// Mitsubishi GX Works2 project: PID_slave_FX3U_26_04_2021   PLC: FX3U/FX3UC

// global labels: Global1
VAR_GLOBAL
  anaDig1 AT D8260 : INT;  (* Analog input from AD converter Level transmitter *)
  anaDig2 AT D8261 : INT;  (* Analog input from AD converter Flow transmitter *)
  digAna AT D8262 : INT;  (* Analog output from DA converter Level Vaulve *)
  Pump AT Y000 : BOOL;  (* Kontaktor til drift av pumpe *)
  AlarmLamp AT Y001 : BOOL;  (* Alarm lampe til systemet *)
  MagnetValve_1 AT Y004 : BOOL;  (* Magnetventil 1 *)
  MagnetValve_2 AT Y005 : BOOL;  (* Magnetventil 2 *)
  MagnetValve_3 AT Y006 : BOOL;  (* Magnetventil 3 *)
  Input_OnOff AT M100 : BOOL;  (* On off for the system *)
  Input_ManualMode AT M500 : BOOL;  (* Valg av Manuell "1" eller Auto "0" *)
  Input_OperationModus AT M501 : BOOL;  (* Valg av direkte "1" eller Revers "0" Regulering *)
  Input_IntegratorModus AT M502 : BOOL;  (* Valg av Integrator virkning på regulator *)
  Input_DerivatorModus AT M503 : BOOL;  (* Valg av Derivator virkning på regulator *)
  Input_Pump AT M504 : BOOL;  (* Start signal til pumpe fra Master *)
  Input_AlarmLamp AT M505 : BOOL;  (* Start signal til Alarm lampe fra Master *)
  Input_MagnetValve_1 AT M506 : BOOL;  (* Start signal til Magnetventil 1 fra Master *)
  Input_MagnetValve_2 AT M507 : BOOL;  (* Start signal til Magnetventil 2 fra Master *)
  Input_MagnetValve_3 AT M508 : BOOL;  (* Start signal til Magnetventil 3 fra Master *)
  Input_SamplingsTime AT D200 : INT;  (* Samplingstid sendt til PID *)
  Output_PID AT D202 : REAL;  (* Utgangs signal sendt ut fra PID *)
  Input_Referance AT D204 : REAL;  (* Referanse verdi sendt til PID *)
  Input_Process AT D206 : REAL;  (* Prosess verdi Sendt til PID *)
  Input_ManualValue AT D208 : REAL;  (* Manuell verdi sendt til PID *)
  Input_NomValue AT D210 : REAL;  (* Nominelt pådrag *)
  Input_MaxPådrag AT D212 : REAL;  (* Max pådrag *)
  Input_MinPådrag AT D214 : REAL;  (* Min pådrag *)
  Input_Skalert_Samplingstid AT D216 : ARRAY [0..1] OF INT;  (* Samplingstid skalert til timer *)
  Input_KpValue AT D218 : REAL;  (* Valg av Kp verdi *)
  Input_TiValue AT D220 : REAL;  (* Valge av Ti verdi *)
  Input_TdValue AT D222 : REAL;  (* Valg av Td verdi *)
  Input_NValue AT D224 : REAL;  (* Valg av N verdi *)
  Input_TtValue AT D226 : REAL;  (* Valg av Tt verdi *)
  Input_FF_TtValue AT D228 : REAL;  (* Valg av Tt verdi til LeadLag blokk *)
  Input_FF_TnValue AT D230 : REAL;  (* Valg av Tn verdi til LeadLag blokk *)
  Input_FF_KLLValue AT D232 : REAL;  (* Valg av KLL verdi til LeadLag blokk *)
  Output_Leadlag AT D234 : REAL;  (* Utgangsignal sendt ut fra LeadLag blokk *)
  Output_Total AT D236 : REAL;  (* Totalt utgangsignal summert *)
  Input_ErrorValue AT D238 : REAL;  (* Beregnet avvik *)
  Input_Flow AT D240 : REAL;  (* Scaled and converted Flow signal in percentage. *)
  Input_AI_Raw1 AT D400 : INT;
  Output_AO_Raw AT D402 : INT;
  Input_AI_Raw2 AT D404 : INT;
  Output_Tank_high AT M600 : BOOL;
  Output_Tank_low AT M601 : BOOL;
  Output_Tank_high_high AT M602 : BOOL;
  Output_Tank_low_low AT M603 : BOOL;
  Input_Acknowledge_normalHigh AT M608 : BOOL;
  Input_Acknowledge_normalLow AT M609 : BOOL;
  Input_Acknowledge_criticalHigh AT M610 : BOOL;
  Input_Acknowledge_criticalLow AT M611 : BOOL;
  Normal_ErrorCheck AT M650 : ARRAY [0..2] OF BOOL;
  Critical_ErrorCheck AT M653 : ARRAY [0..2] OF BOOL;
  Normal_FaultSignal AT M656 : BOOL;
  Criticall_FaultSignal AT M657 : BOOL;
  Output_NoFault AT M658 : BOOL;
  Output_Normal_ErrorSignal AT M604 : BOOL;
  Output_Critical_ErrorSignal AT M605 : BOOL;
  Output_Power_failure AT M606 : BOOL;
  Input_Acknowledge_powerFailure AT M612 : BOOL;
  Input_Acknowledge_Normal_Error AT M613 : BOOL;
  Input_Acknowledge_Critical_Error AT M614 : BOOL;
  Tank_criticalHigh AT M659 : BOOL;
  Tank_criticalLow AT M660 : BOOL;
  Tank_normalHigh AT M661 : BOOL;
  Tank_normalLow AT M662 : BOOL;
  Tank_normalError AT M663 : BOOL;
  Tank_CriticalError AT M664 : BOOL;
  Input_PID_ON AT M509 : BOOL;  (* On Off switch for PID Function block *)
  Input_LeadLag1_ON AT M510 : BOOL;  (* On Off switch for Leadlag function block1 *)
  Input_LeadLag2_ON AT M511 : BOOL;  (* On Off switch for Leadlag function block 2 *)
  Output_Profibus_error_signal AT M512 : BOOL;
  Master_Power_failure AT M513 : BOOL;
END_VAR

// task Task_01 (event TRUE, interval 0, priority 31): POU_01

FUNCTION_BLOCK Filter_Midling
VAR_INPUT
  Filter_Input : DINT;  (* Inngangs verdi til filter *)
END_VAR
VAR
  Filter_Array : ARRAY [0..39] OF DINT;  (* Array av inngangsverdier *)
END_VAR
VAR_INPUT
  Enable : BOOL;  (* Enabler *)
END_VAR
VAR
  Filter_CalcSum : DINT;  (* Calc of output *)
  Filter_Divided : DINT;  (* Utgangsverdi til filter *)
END_VAR
VAR_OUTPUT
  Filter_Output : INT;
END_VAR
VAR
  Index : INT;
END_VAR
VAR_INPUT
  Filter_Degree : INT;  (* Inngangs verdi til filter *)
END_VAR
IF ENABLE THEN
	Filter_Array[0] := Filter_Input;
	

	Filter_CalcSum:=  0;
	FOR Index:= 0 TO (Filter_Degree-1) DO 
		Filter_CalcSum :=  Filter_CalcSum + Filter_Array[Index];
	END_FOR;
	
	Filter_Divided:= Filter_CalcSum/int_to_dint(Filter_Degree);
	
	Filter_Output:= DINT_TO_INT(Filter_Divided);
	
	FOR Index := 0 TO (Filter_Degree -2 ) DO 
		Filter_Array[(Filter_Degree-1)-Index] := Filter_Array[(Filter_Degree-2) -Index];
	END_FOR;
		

ELSE
	;
END_IF;
END_FUNCTION_BLOCK

FUNCTION_BLOCK LeadLag
VAR_INPUT
  LeadLag_Enable : BOOL;  (* Enable for hvert samplingstid *)
  LeadLag_Samplingstid : INT;  (* Samplingstid Lead Lag blokk *)
  LeadLag_InputValue : REAL;  (* Inngangsverdi inn til LeadLag blokk *)
  LeadLag_Tt : REAL;  (* Tt konstant for Lead Lag blokk *)
  LeadLag_Tn : REAL;  (* Tn konstant for Lead Lag blokk *)
  LeadLag_KLL : REAL;  (* KLL konstant for Lead Lag blokk *)
END_VAR
VAR_OUTPUT
  LeadLag_Output : REAL;  (* Utgangsverdu ut fra LeadLag blokk *)
END_VAR
VAR
  LeadLag_Mellomregning_Sampl : REAL;  (* Mellom regning for samplingstid *)
  LeadLag_Skalert_Samplingstid : REAL;  (* Skalert samplingstid i sekunder *)
  LeadLag_InputValue_F : ARRAY [0..1] OF REAL;  (* Input verdi denne og forrige *)
  LeadLag_Output_F : ARRAY [0..1] OF REAL;  (* Utgangspådrag  (denne og forrige) *)
END_VAR
(*Omgjøring av samplingstid fra ms til s*)
FLT(TRUE , leadlag_Samplingstid, leadLag_Mellomregning_Sampl);
LeadLag_Skalert_Samplingstid := leadlag_Mellomregning_Sampl/1000.0;

IF LeadLag_Enable THEN
	LeadLag_InputValue_F[0] := LeadLag_InputValue;
	
	LeadLag_Output_F[0] := (LeadLag_KLL*((LeadLag_Tt+LeadLag_Skalert_Samplingstid)*LeadLag_InputValue_F[0]-LeadLag_Tt*LeadLag_InputValue_F[1])+LeadLag_Tn*LeadLag_Output_F[1])/(LeadLag_Tn+LeadLag_Skalert_Samplingstid);
	
	LeadLag_Output_F[1] := LeadLag_Output_F[0];
	LeadLag_InputValue_F[1] := LeadLag_InputValue_F[0];
	
	LeadLag_Output := LeadLag_Output_F[0];
ELSE

;
END_IF;


;
END_FUNCTION_BLOCK

FUNCTION_BLOCK My_PID
VAR_INPUT
  PID_Enable : BOOL;  (* Samplings enable *)
  PID_Referanse : REAL;  (* Referanseverdi PID blokk *)
  PID_ProcessValue : REAL;  (* Prosessverdi PID blokk *)
  PID_Samplingstime : INT;  (* Samplingstid PID blokk (ms) *)
  PID_Kp : REAL;  (* KP PID blokk *)
  PID_Ti : REAL;  (* Ti PID blokk *)
  PID_Td : REAL;  (* Td PID blokk *)
  PID_N : REAL;  (* Filter konstant for Tf *)
  PID_Tt : REAL;  (* Tracking konstant for PID tracking inngang *)
  PID_IntegralMode : BOOL;  (* Integrator for PID blokk *)
  PID_DerivatorMode : BOOL;  (* Derivator for PID blokk *)
  PID_OperationMode : BOOL;  (* Direkte kobling "1", reversert "0" *)
  PID_ManualMode : BOOL;  (* Auto "0" , Manuell pådrag "1" *)
  PID_ManualValue : REAL;  (* Manuelt pådrag verdi *)
END_VAR
VAR_IN_OUT
  PID_NomValue : REAL;  (* Nominelt pådrags verdi *)
END_VAR
VAR_INPUT
  PID_MaxOutput : REAL;  (* Max pådrags verdi *)
  PID_MinOutput : REAL;  (* Min pådrags verdi *)
END_VAR
VAR_OUTPUT
  PID_Output : REAL;  (* Utgangsverdi fra PID-reg *)
  PID_ErrorValue : REAL;  (* Error value from PID-regulator *)
END_VAR
VAR
  PID_Alpha : REAL;  (* Beregnet alpha verdi *)
  PID_Beta : REAL;  (* Beregnet betaverdi *)
  PID_Gamma : REAL;  (* Beregnet gammaverdi *)
  PID_ErrorValue_F : ARRAY [0..1] OF REAL;  (* Beregnet error verdi (Denne og forrige verdi) *)
  PID_PGain : ARRAY [0..1] OF REAL;  (* Beregnet P forsterkning (Denne og forrige verdi) *)
  PID_IGain : ARRAY [0..1] OF REAL;  (* Beregnet I forsterkning (Denne og forrige verdi) *)
  PID_DGain : ARRAY [0..1] OF REAL;  (* Beregnet D forsterkning (Denne og forrige verdi) *)
  PID_Gain_Total : REAL;  (* Beregnet sum av total pådrag (Ubegrenset verdi) *)
  PID_Gain_Tracking : REAL;  (* Beregnet sum av tracking pådrag (Begrenset verdi) *)
  PID_ProcessValue_F : ARRAY [0..1] OF REAL;  (* Prosess verdi i PID blokk (denne og forrige verdi) *)
  PID_Scaled_Samplingstime : REAL;  (* Skalert samplingstid i sekunder *)
  PID_Calc_Sampling : REAL;  (* Mellomregning av samplingstid *)
  Regulatortype : ARRAY [0..1] OF INT;  (* Array to know current and last regulator type *)
END_VAR
(*Omgjøring av samplingstid fra ms til s*)
FLT(TRUE , PID_Samplingstime, PID_Calc_Sampling);
PID_Scaled_Samplingstime := PID_Calc_Sampling/1000.0;



(*Systemet vil gå inn i koden hvert samplingstid som er satt*)

IF PID_Enable THEN	
	
	
	(*Regning av konstanter alpha, beta, gamma og lagring av prosessverdi til et array*)
	PID_Alpha := PID_Scaled_Samplingstime/PID_Ti;
	PID_Beta := PID_Td/(PID_Td + (PID_Scaled_Samplingstime*pid_n));
	PID_ProcessValue_F[0] := PID_ProcessValue;
	
	IF PID_Tt > 0.0 THEN 
		PID_Gamma:= PID_Scaled_Samplingstime/PID_Tt;
	ELSE
		PID_Gamma:= 0.0;
	END_IF;

	(*IF statement to differentiate between the regulator types:		0 = P-reg.	1 = PD-reg.	2 = PI-reg.	3 = PID-reg*)
	IF PID_IntegralMode AND PID_DerivatorMode THEN
		Regulatortype[0] := 3; (*PID-regulator*)													
	ELSIF PID_IntegralMode AND NOT PID_DerivatorMode THEN
		Regulatortype[0] := 2; (*PI-regulator*)
	ELSIF PID_DerivatorMode AND NOT PID_IntegralMode THEN
		Regulatortype[0] := 1; (*PD-regulator*)
	ELSE
		Regulatortype[0] := 0; (*P-regulator*) 
	END_IF;
	
	(*IF statement that sets PID_IGain[0] to PID_NomValue if switching from P to PI or PID reg. when nominal value is not 0.0, and PID_IGain[0] to 0.0 if switching from P to PI or PID reg. when nominal value = 0.0.*)
	(*This prevents leaps in the PID_output value when switching to a regulator with integral gain.*)
	IF PID_NomValue <> 0.0 AND Regulatortype[0] = 2 AND Regulatortype[1] = 0 OR PID_NomValue <> 0.0 AND Regulatortype[0] = 3 AND Regulatortype[1] = 0 THEN
		PID_IGain[0] := PID_NomValue;
	ELSIF PID_NomValue = 0.0 AND Regulatortype[0] = 2 AND Regulatortype[1] = 0 OR  PID_NomValue = 0.0 AND Regulatortype[0] = 3 AND Regulatortype[1] = 0 THEN
		PID_IGain[0] := 0.0;
	END_IF;
	
	(*IF statement that sets PID_IGain[0] to PID_NomValue if switching from PD to PI or PID reg. when nominal value is not 0.0, and PID_IGain[0] to 0.0 if switching from PD to PI or PID reg. when nominal value = 0.0.*)
	(*This prevents leaps in the PID_output value when switching to a regulator with integral gain.*)
	IF PID_NomValue <> 0.0 AND Regulatortype[0] = 2 AND Regulatortype[1] = 1 OR PID_NomValue <> 0.0 AND Regulatortype[0] = 3 AND Regulatortype[1] = 1 THEN
		PID_IGain[0] := PID_NomValue;
	ELSIF PID_NomValue = 0.0 AND Regulatortype[0] = 2 AND Regulatortype[1] = 1 OR  PID_NomValue = 0.0 AND Regulatortype[0] = 3 AND Regulatortype[1] = 1 THEN
		PID_IGain[0] := 0.0;
	END_IF;
	
	(*IF statement that prevents leaps in the PID_output value when sitching to a regulator without integral gain*)
	IF Regulatortype[0] = 0 AND Regulatortype[1] = 2 OR  Regulatortype[0] = 0 AND Regulatortype[1] = 3 THEN
		PID_NomValue:= PID_IGain[0]+PID_NomValue;
	END_IF;
	
	(*IF statement that prevents leaps in the PID_output value when sitching to a regulator without integral gain*)
	IF Regulatortype[0] = 1 AND Regulatortype[1] = 2 OR  Regulatortype[0] = 1 AND Regulatortype[1] = 3 THEN
		PID_NomValue:= PID_IGain[0]+PID_NomValue;
	END_IF;
	
	(*Leaps in the PID_output value when sitching to a regulator with derivative gain is prevented by swithing when the system is stable. Same is applicaple when switching to a regulator without derivative gain.*)
	
	Regulatortype[1] := Regulatortype[0]; (*Last regulator type stored in variable*)


	
	(*Regning av avvik mtp om det er direkte eller revers regulering*)
	IF PID_OperationMode THEN
		PID_ErrorValue_F[0] := PID_ProcessValue_F[0] - PID_Referanse;
	ELSE
		PID_ErrorValue_F[0] := PID_Referanse - PID_ProcessValue_F[0];
	END_IF;
	

	(*Beregning av pådragsbidrag fra P-del*)
	PID_PGain[0] := PID_Kp*PID_ErrorValue_F[0];
	
	(*Ser om integrator er aktivert og beregner pådragsbidrag fra I-del med tracking inngang*)
	IF PID_IntegralMode THEN
		PID_IGain[0] := PID_IGain[1] + PID_Kp*PID_Alpha*PID_ErrorValue_F[0]+PID_Gamma*(PID_Gain_Tracking-PID_Gain_Total);
	ELSE
		PID_IGain[0] := 0.0;
	END_IF;
	
	(*Ser om Derivator er aktivert og beregner pådragsbidrag fra D-del*)
	IF PID_DerivatorMode THEN
		PID_DGain[0] := (PID_Beta*PID_DGain[1]) - ((PID_Kp*PID_Td/PID_Scaled_Samplingstime)*(1.0-PID_Beta)*(PID_ProcessValue_F[0]-PID_ProcessValue_F[1]));
	ELSE 
		PID_DGain[0] := 0.0;
	END_IF;
	
	(*Summerer sammen pådragsbidrag fra alle delene*)
	PID_Gain_Total := PID_PGain[0] + PID_IGain[0] + PID_DGain[0] + PID_NomValue;
	
	(*Oppdatering av verdier*)
	PID_ErrorValue_F[1] := PID_ErrorValue_F[0];
	PID_ProcessValue_F[1] := PID_ProcessValue_F[0];
	PID_PGain[1] := PID_PGain[0];
	PID_IGain[1] := PID_IGain[0];
	PID_DGain[1] := PID_DGain[0];
	
	(*Ser om regulatoren skal gå i auto eller manuell modus*)
	IF PID_ManualMode THEN 
		PID_Gain_Tracking := PID_ManualValue;
	ELSE 
		PID_Gain_Tracking := PID_Gain_Total;
	END_IF;
	
	(*Kontrollerer at pådragsbidrag er innenfor min og max verdier*)
	IF PID_Gain_Tracking > PID_maxoutput THEN
		PID_Gain_Tracking:= PID_MaxOutput ;
	ELSIF PID_Gain_Tracking< PID_MinOutput THEN 
		PID_Gain_Tracking:= PID_MinOutput;
	ELSE
		PID_Gain_Tracking:= PID_Gain_Tracking;
	END_IF;
	
	(*Utgang fra PID regulator*)
	PID_Output := PID_Gain_Tracking;
	PID_ErrorValue:= PID_ErrorValue_F[0];
ELSE 
;
END_IF;
END_FUNCTION_BLOCK

FUNCTION_BLOCK Output_Adder
VAR_INPUT
  Adder_Enable : BOOL;
  Adder_Input1 : REAL;  (* Input value 1 *)
  Adder_Input2 : REAL;  (* Input value 2 *)
  Adder_Input3 : REAL;  (* Input value 3 *)
  Adder_Input4 : REAL;  (* Input value 4 *)
  Adder_Input5 : REAL;  (* Input value 5 *)
  Adder_HighLimit : REAL;  (* Maximum output *)
  Adder_LowLimit : REAL;  (* Minimum output *)
END_VAR
VAR_OUTPUT
  Adder_Output : REAL;  (* Total output from adder *)
END_VAR
VAR
  Adder_Sum : REAL;  (* Sum av inputs *)
END_VAR
IF Adder_Enable THEN
	Adder_Sum := Adder_Input1+Adder_Input2+Adder_Input3+Adder_Input4+Adder_Input5;
	
	IF Adder_Sum > Adder_HighLimit THEN
		Adder_Output := Adder_HighLimit;
	ELSIF Adder_Sum < Adder_LowLimit THEN
		Adder_Output := Adder_LowLimit;
	ELSE
		Adder_Output := Adder_Sum;
	END_IF;
END_IF;
;
END_FUNCTION_BLOCK

PROGRAM POU_01
VAR
  My_PID_1 : My_PID;
  LeadLag_1 : LeadLag;
  Output_Adder_1 : Output_Adder;
  Filter_Midling_1 : Filter_Midling;
  Filter_Midling_2 : Filter_Midling;
END_VAR
(* structured ladder/FBD written out as ST: instructions are called as NAME(EN, inputs, outputs); _pN, _eN, _tN stand for wires *)
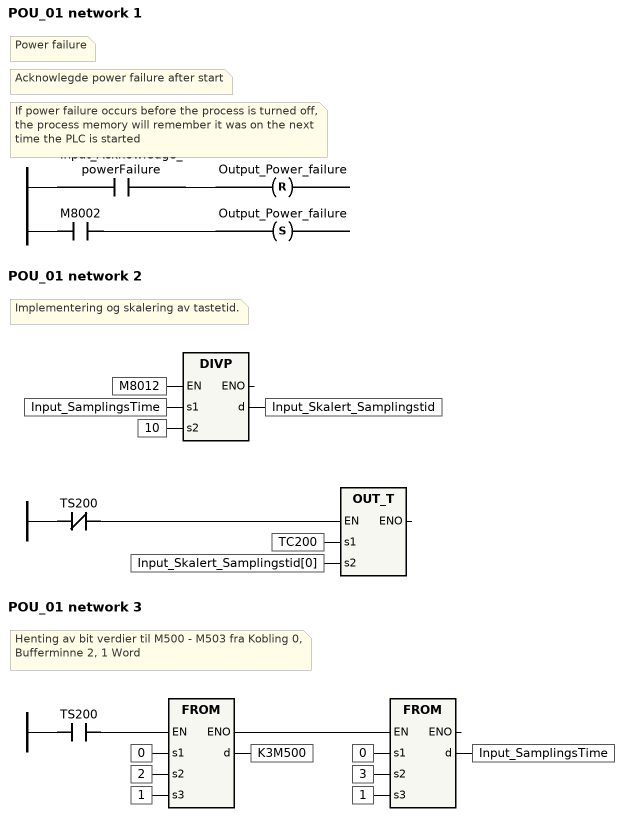
(* network 1 *)
(* Power failure *)
(* Acknowlegde power failure after start *)
(* If power failure occurs before the process is turned off, the process memory will remember it was on the next time the PLC is started *)
RST(Input_Acknowledge_powerFailure, Output_Power_failure);
SET(M8002, Output_Power_failure);
(* network 2 *)
(* Implementering og skalering av tastetid. *)
DIVP(M8012, Input_SamplingsTime, 10, Input_Skalert_Samplingstid);
OUT_T(NOT TS200, TC200, Input_Skalert_Samplingstid[0]);
(* network 3 *)
(* Henting av bit verdier til M500 - M503 fra Kobling 0, Bufferminne 2, 1 Word *)
_e1 := FROM(TS200, 0, 2, 1, K3M500);
FROM(_e1, 0, 3, 1, Input_SamplingsTime);
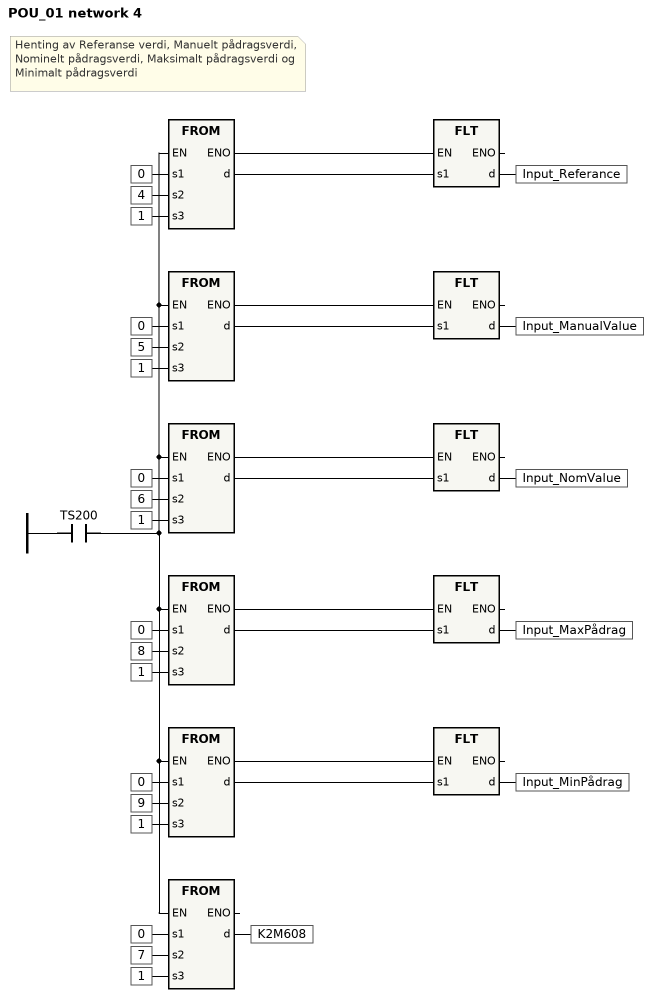
(* network 4 *)
(* Henting av Referanse verdi, Manuelt pådragsverdi, Nominelt pådragsverdi, Maksimalt pådragsverdi og Minimalt pådragsverdi *)
_e2 := FROM(TS200, 0, 4, 1, _t1);
FLT(_e2, _t1, Input_Referance);
_e4 := FROM(TS200, 0, 5, 1, _t3);
FLT(_e4, _t3, Input_ManualValue);
_e6 := FROM(TS200, 0, 6, 1, _t5);
FLT(_e6, _t5, Input_NomValue);
FROM(TS200, 0, 7, 1, K2M608);
_e8 := FROM(TS200, 0, 8, 1, _t7);
FLT(_e8, _t7, Input_MaxPådrag);
_e10 := FROM(TS200, 0, 9, 1, _t9);
FLT(_e10, _t9, Input_MinPådrag);
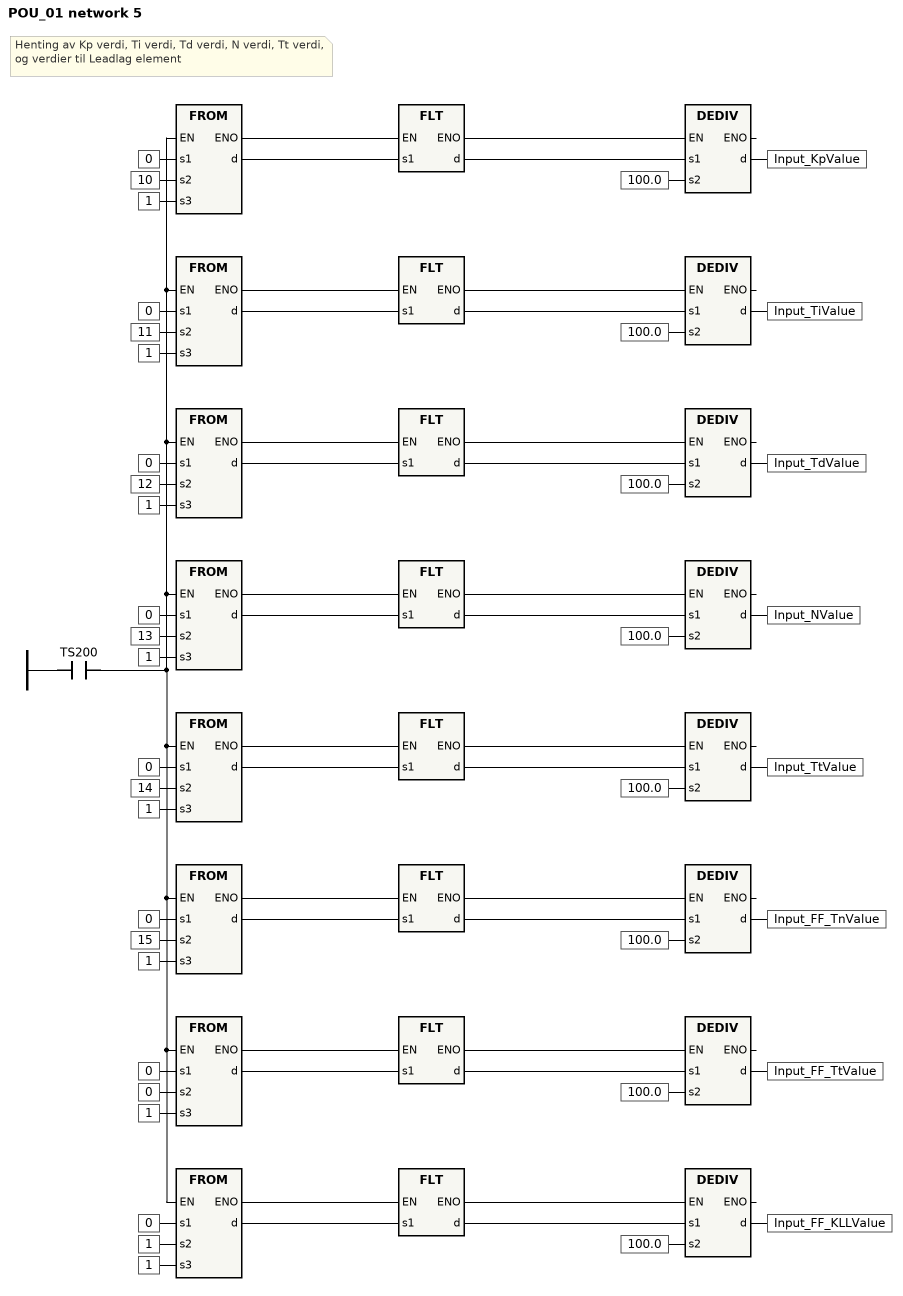
(* network 5 *)
(* Henting av Kp verdi, Ti verdi, Td verdi, N verdi, Tt verdi, og verdier til Leadlag element *)
_e2 := FROM(TS200, 0, 10, 1, _t1);
_e4 := FLT(_e2, _t1, _t3);
DEDIV(_e4, _t3, 100.0, Input_KpValue);
_e6 := FROM(TS200, 0, 11, 1, _t5);
_e8 := FLT(_e6, _t5, _t7);
DEDIV(_e8, _t7, 100.0, Input_TiValue);
_e10 := FROM(TS200, 0, 12, 1, _t9);
_e12 := FLT(_e10, _t9, _t11);
DEDIV(_e12, _t11, 100.0, Input_TdValue);
_e14 := FROM(TS200, 0, 13, 1, _t13);
_e16 := FLT(_e14, _t13, _t15);
DEDIV(_e16, _t15, 100.0, Input_NValue);
_e18 := FROM(TS200, 0, 14, 1, _t17);
_e20 := FLT(_e18, _t17, _t19);
DEDIV(_e20, _t19, 100.0, Input_TtValue);
_e22 := FROM(TS200, 0, 15, 1, _t21);
_e24 := FLT(_e22, _t21, _t23);
DEDIV(_e24, _t23, 100.0, Input_FF_TnValue);
_e26 := FROM(TS200, 0, 0, 1, _t25);
_e28 := FLT(_e26, _t25, _t27);
DEDIV(_e28, _t27, 100.0, Input_FF_TtValue);
_e30 := FROM(TS200, 0, 1, 1, _t29);
_e32 := FLT(_e30, _t29, _t31);
DEDIV(_e32, _t31, 100.0, Input_FF_KLLValue);
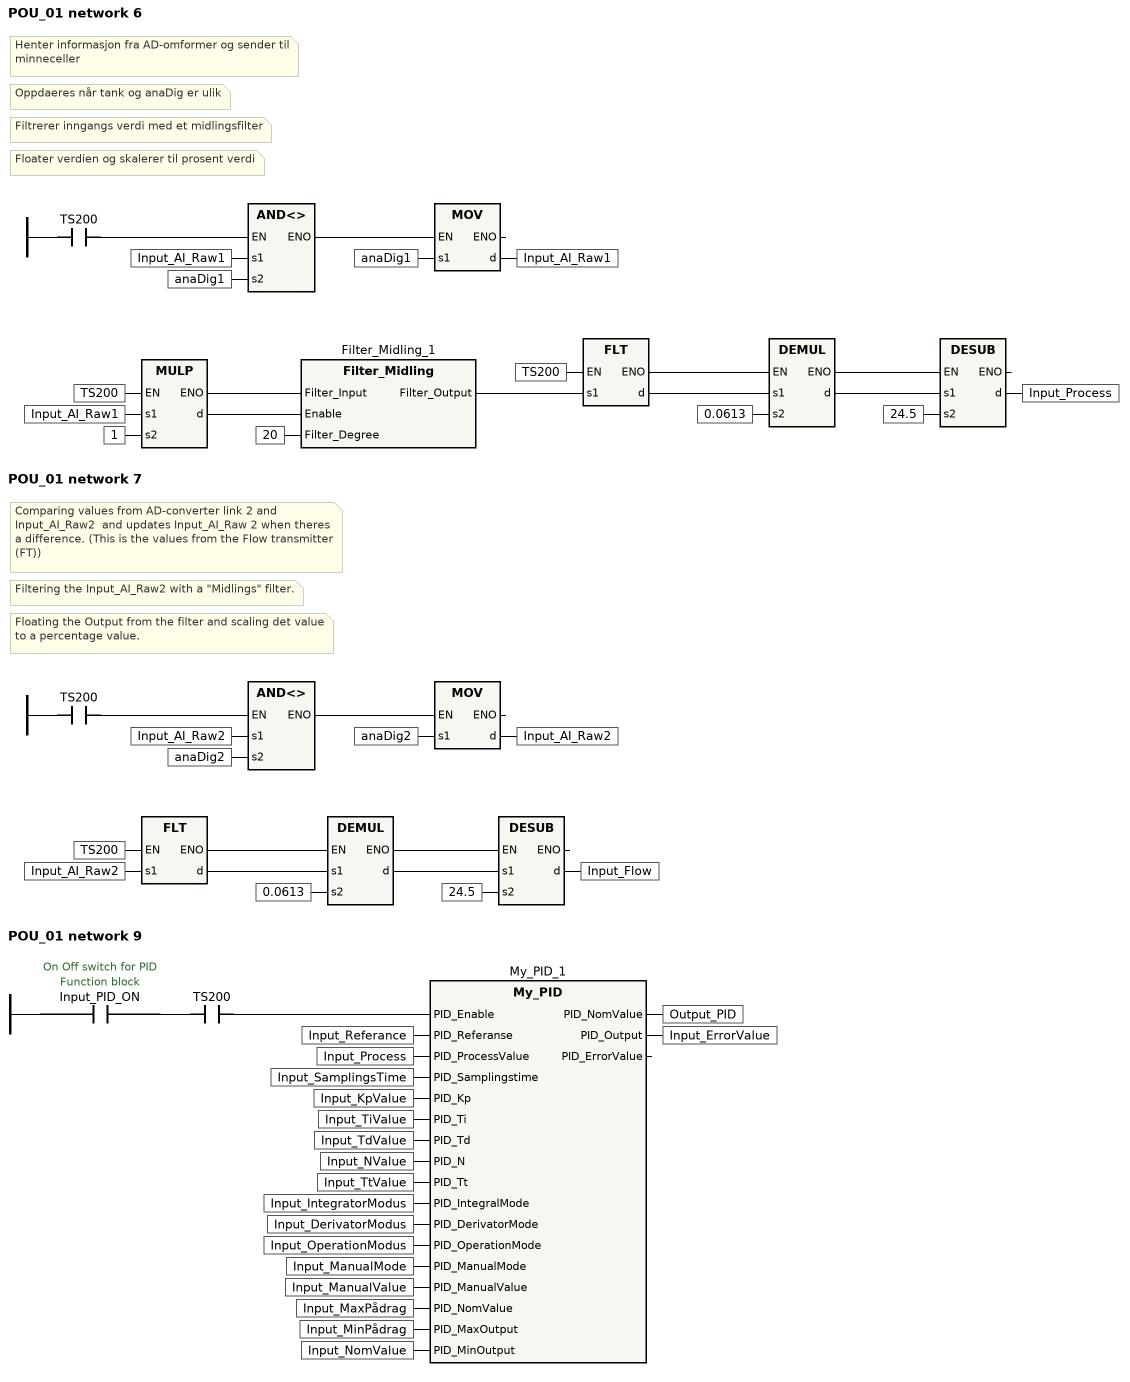
(* network 6 *)
(* Henter informasjon fra AD-omformer og sender til minneceller *)
(* Oppdaeres når tank og anaDig er ulik *)
(* Filtrerer inngangs verdi med et midlingsfilter *)
(* Floater verdien og skalerer til prosent verdi *)
_e1 := AND<>(TS200, Input_AI_Raw1, anaDig1);
MOV(_e1, anaDig1, Input_AI_Raw1);
_e3 := MULP(TS200, Input_AI_Raw1, 1, _t2);
Filter_Midling_1(Filter_Input := _e3, Enable := _t2, Filter_Degree := 20);
_e5 := FLT(TS200, Filter_Midling_1.Filter_Output, _t4);
_e7 := DEMUL(_e5, _t4, 0.0613, _t6);
DESUB(_e7, _t6, 24.5, Input_Process);
(* network 7 *)
(* Comparing values from AD-converter link 2 and Input_AI_Raw2  and updates Input_AI_Raw 2 when theres a difference. (This is the values from the Flow transmitter (FT)) *)
(* Filtering the Input_AI_Raw2 with a "Midlings" filter. *)
(* Floating the Output from the filter and scaling det value to a percentage value. *)
_e1 := AND<>(TS200, Input_AI_Raw2, anaDig2);
MOV(_e1, anaDig2, Input_AI_Raw2);
_e3 := FLT(TS200, Input_AI_Raw2, _t2);
_e5 := DEMUL(_e3, _t2, 0.0613, _t4);
DESUB(_e5, _t4, 24.5, Input_Flow);
(* network 9 *)
My_PID_1(PID_Enable := Input_PID_ON AND TS200, PID_Referanse := Input_Referance, PID_ProcessValue := Input_Process, PID_Samplingstime := Input_SamplingsTime, PID_Kp := Input_KpValue, PID_Ti := Input_TiValue, PID_Td := Input_TdValue, PID_N := Input_NValue, PID_Tt := Input_TtValue, PID_IntegralMode := Input_IntegratorModus, PID_DerivatorMode := Input_DerivatorModus, PID_OperationMode := Input_OperationModus, PID_ManualMode := Input_ManualMode, PID_ManualValue := Input_ManualValue, PID_NomValue := Input_MaxPådrag, PID_MaxOutput := Input_MinPådrag, PID_MinOutput := Input_NomValue, PID_Output => Input_ErrorValue);
Output_PID := My_PID_1.PID_NomValue;
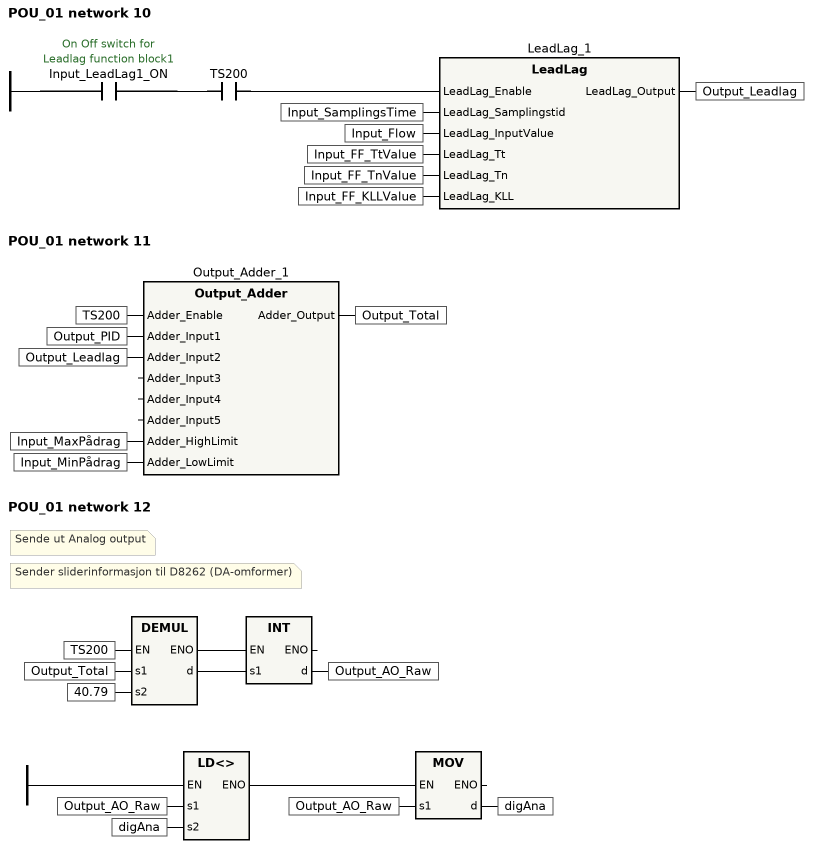
(* network 10 *)
LeadLag_1(LeadLag_Enable := Input_LeadLag1_ON AND TS200, LeadLag_Samplingstid := Input_SamplingsTime, LeadLag_InputValue := Input_Flow, LeadLag_Tt := Input_FF_TtValue, LeadLag_Tn := Input_FF_TnValue, LeadLag_KLL := Input_FF_KLLValue, LeadLag_Output => Output_Leadlag);
(* network 11 *)
Output_Adder_1(Adder_Enable := TS200, Adder_Input1 := Output_PID, Adder_Input2 := Output_Leadlag, Adder_HighLimit := Input_MaxPådrag, Adder_LowLimit := Input_MinPådrag, Adder_Output => Output_Total);
(* network 12 *)
(* Sende ut Analog output *)
(* Sender sliderinformasjon til D8262 (DA-omformer) *)
_e2 := DEMUL(TS200, Output_Total, 40.79, _t1);
INT(_e2, _t1, Output_AO_Raw);
_e3 := LD<>(TRUE, Output_AO_Raw, digAna);
MOV(_e3, Output_AO_Raw, digAna);
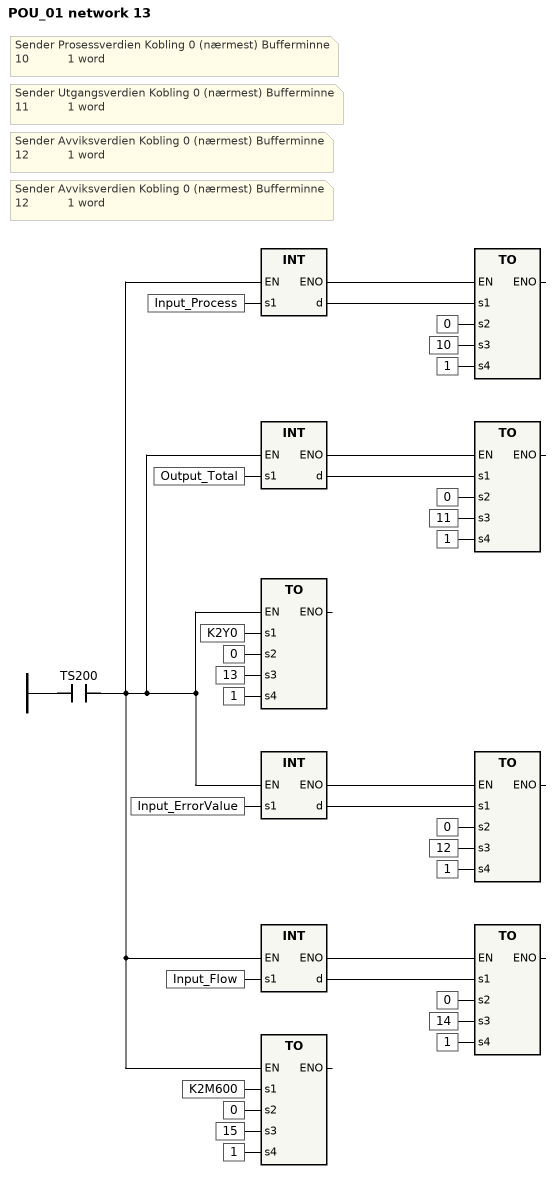
(* network 13 *)
(* Sender Prosessverdien Kobling 0 (nærmest) Bufferminne 10           1 word *)
(* Sender Utgangsverdien Kobling 0 (nærmest) Bufferminne 11           1 word *)
(* Sender Avviksverdien Kobling 0 (nærmest) Bufferminne 12           1 word *)
(* Sender Avviksverdien Kobling 0 (nærmest) Bufferminne 12           1 word *)
_e2 := INT(TS200, Input_Process, _t1);
TO(_e2, _t1, 0, 10, 1);
_e4 := INT(TS200, Output_Total, _t3);
TO(_e4, _t3, 0, 11, 1);
_e6 := INT(TS200, Input_ErrorValue, _t5);
TO(_e6, _t5, 0, 12, 1);
TO(TS200, K2Y0, 0, 13, 1);
_e8 := INT(TS200, Input_Flow, _t7);
TO(_e8, _t7, 0, 14, 1);
TO(TS200, K2M600, 0, 15, 1);
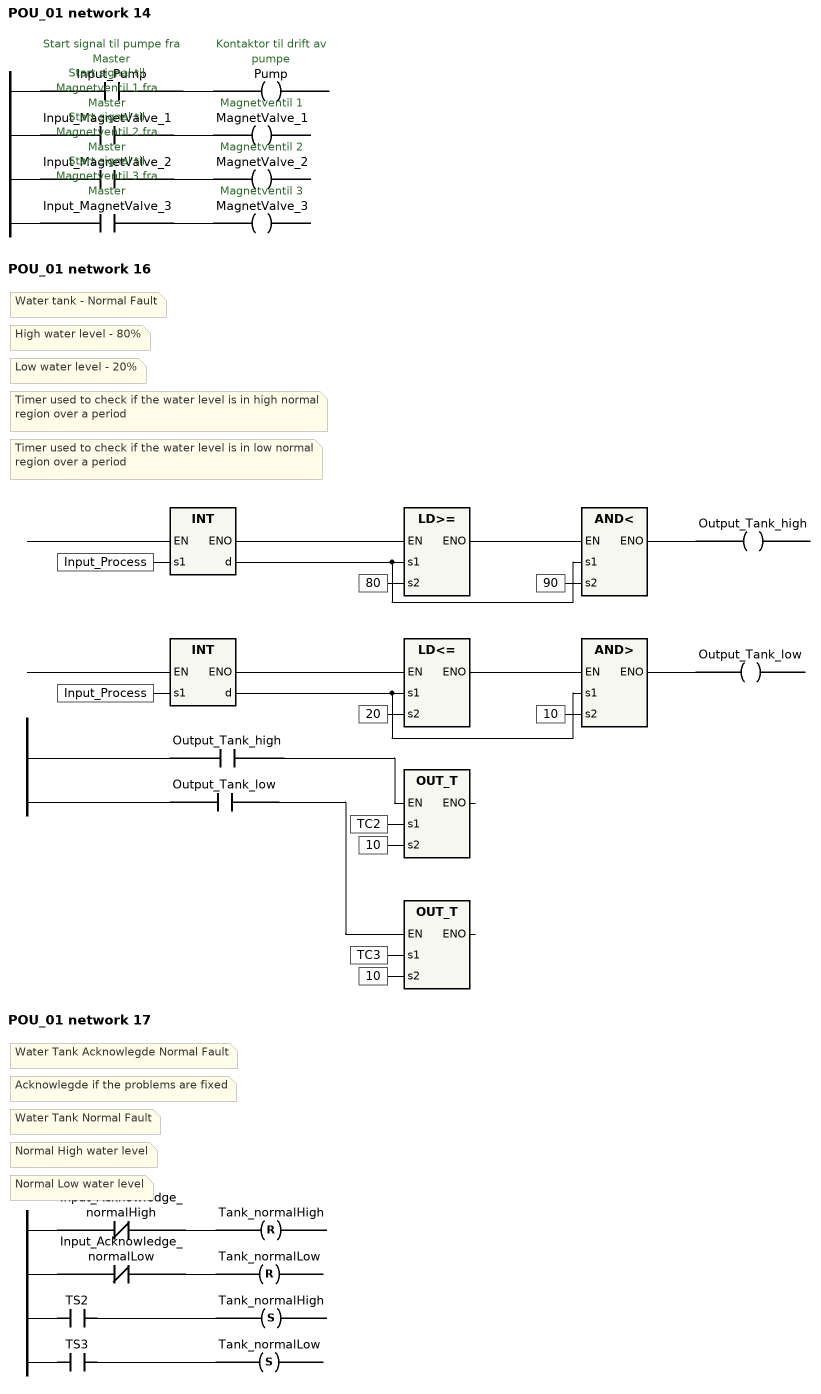
(* network 14 *)
Pump := Input_Pump;
MagnetValve_1 := Input_MagnetValve_1;
MagnetValve_2 := Input_MagnetValve_2;
MagnetValve_3 := Input_MagnetValve_3;
(* network 16 *)
(* Water tank - Normal Fault *)
(* High water level - 80% *)
(* Low water level - 20% *)
(* Timer used to check if the water level is in high normal region over a period *)
(* Timer used to check if the water level is in low normal region over a period *)
_e2 := INT(TRUE, Input_Process, _t1);
_e3 := LD>=(_e2, _t1, 80);
_e4 := AND<(_e3, _t1, 90);
Output_Tank_high := _e4;
_e6 := INT(TRUE, Input_Process, _t5);
_e7 := LD<=(_e6, _t5, 20);
_e8 := AND>(_e7, _t5, 10);
Output_Tank_low := _e8;
OUT_T(Output_Tank_high, TC2, 10);
OUT_T(Output_Tank_low, TC3, 10);
(* network 17 *)
(* Water Tank Acknowlegde Normal Fault *)
(* Acknowlegde if the problems are fixed *)
(* Water Tank Normal Fault *)
(* Normal High water level *)
(* Normal Low water level *)
RST(NOT Input_Acknowledge_normalHigh, Tank_normalHigh);
RST(NOT Input_Acknowledge_normalLow, Tank_normalLow);
SET(TS2, Tank_normalHigh);
SET(TS3, Tank_normalLow);
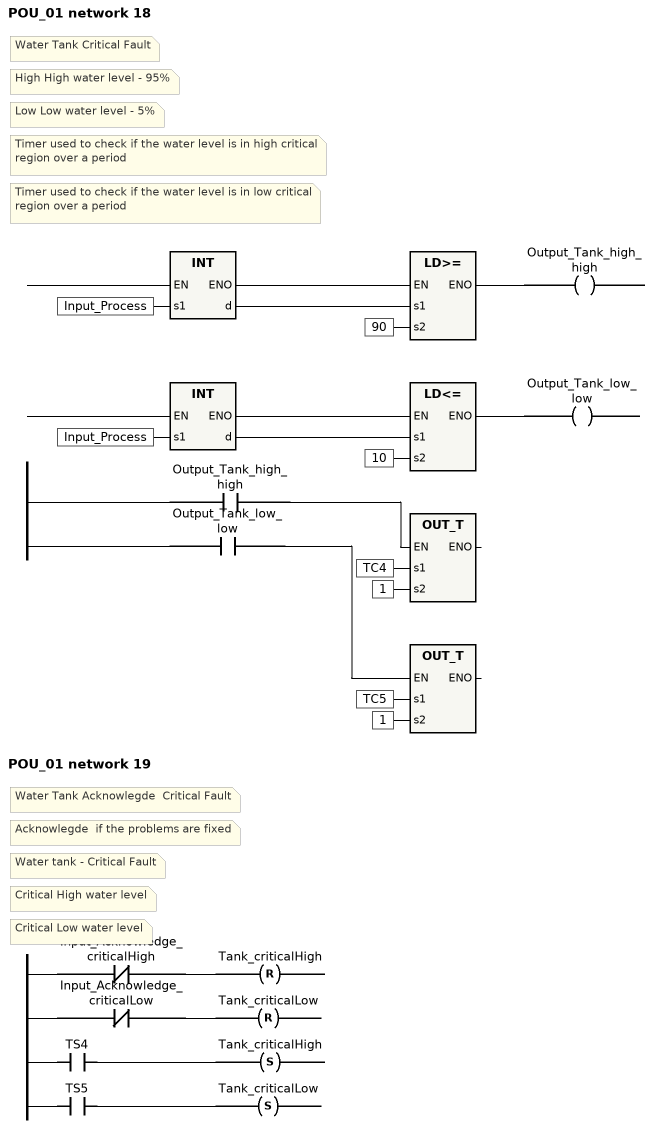
(* network 18 *)
(* Water Tank Critical Fault *)
(* High High water level - 95% *)
(* Low Low water level - 5% *)
(* Timer used to check if the water level is in high critical region over a period *)
(* Timer used to check if the water level is in low critical region over a period *)
_e2 := INT(TRUE, Input_Process, _t1);
_e3 := LD>=(_e2, _t1, 90);
Output_Tank_high_high := _e3;
_e5 := INT(TRUE, Input_Process, _t4);
_e6 := LD<=(_e5, _t4, 10);
Output_Tank_low_low := _e6;
OUT_T(Output_Tank_high_high, TC4, 1);
OUT_T(Output_Tank_low_low, TC5, 1);
(* network 19 *)
(* Water Tank Acknowlegde  Critical Fault *)
(* Acknowlegde  if the problems are fixed *)
(* Water tank - Critical Fault *)
(* Critical High water level *)
(* Critical Low water level *)
RST(NOT Input_Acknowledge_criticalHigh, Tank_criticalHigh);
RST(NOT Input_Acknowledge_criticalLow, Tank_criticalLow);
SET(TS4, Tank_criticalHigh);
SET(TS5, Tank_criticalLow);
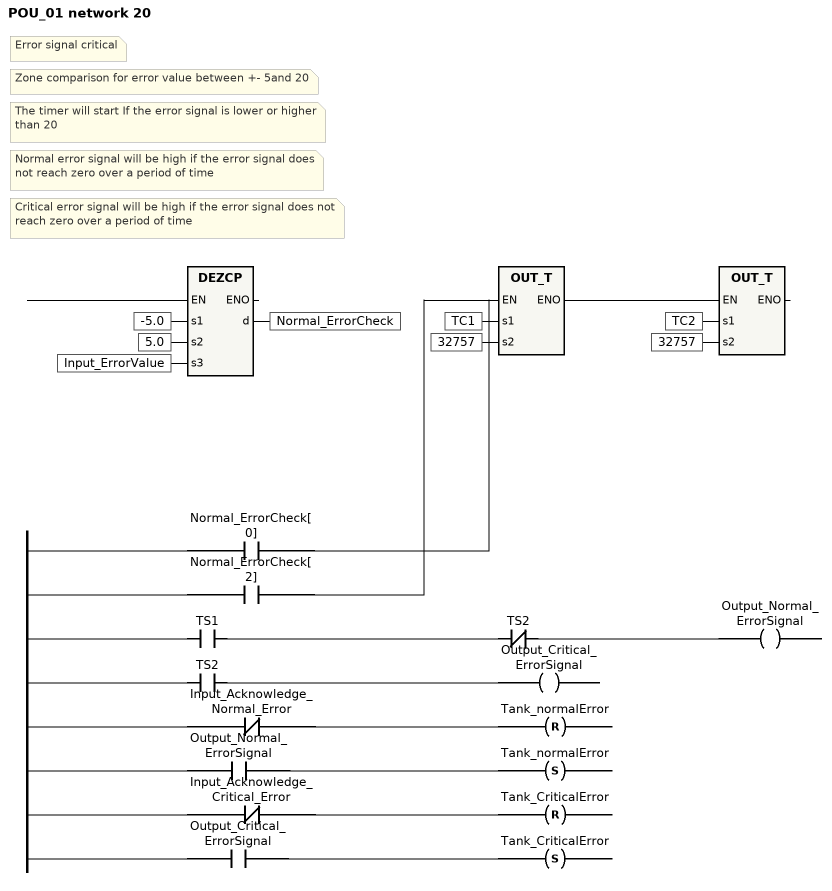
(* network 20 *)
(* Error signal critical *)
(* Zone comparison for error value between +- 5and 20 *)
(* The timer will start If the error signal is lower or higher than 20 *)
(* Normal error signal will be high if the error signal does not reach zero over a period of time *)
(* Critical error signal will be high if the error signal does not reach zero over a period of time *)
DEZCP(TRUE, -5.0, 5.0, Input_ErrorValue, Normal_ErrorCheck);
_e1 := OUT_T(Normal_ErrorCheck[0] OR Normal_ErrorCheck[2], TC1, 32757);
OUT_T(_e1, TC2, 32757);
Output_Normal_ErrorSignal := TS1 AND NOT TS2;
Output_Critical_ErrorSignal := TS2;
RST(NOT Input_Acknowledge_Normal_Error, Tank_normalError);
SET(Output_Normal_ErrorSignal, Tank_normalError);
RST(NOT Input_Acknowledge_Critical_Error, Tank_CriticalError);
SET(Output_Critical_ErrorSignal, Tank_CriticalError);
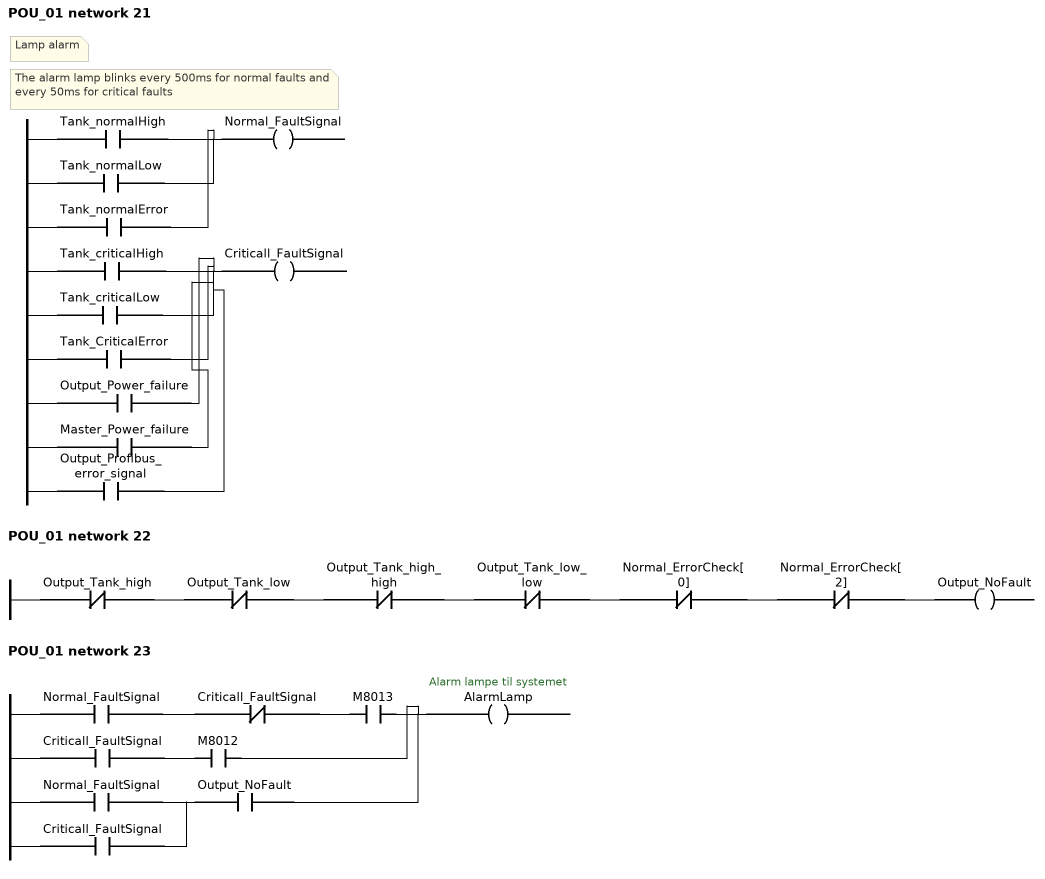
(* network 21 *)
(* Lamp alarm *)
(* The alarm lamp blinks every 500ms for normal faults and every 50ms for critical faults *)
Normal_FaultSignal := Tank_normalHigh OR Tank_normalLow OR Tank_normalError;
Criticall_FaultSignal := Tank_criticalHigh OR Tank_criticalLow OR Tank_CriticalError OR Output_Power_failure OR Master_Power_failure OR Output_Profibus_error_signal;
(* network 22 *)
Output_NoFault := NOT Output_Tank_high AND NOT Output_Tank_low AND NOT Output_Tank_high_high AND NOT Output_Tank_low_low AND NOT Normal_ErrorCheck[0] AND NOT Normal_ErrorCheck[2];
(* network 23 *)
AlarmLamp := (Normal_FaultSignal AND NOT Criticall_FaultSignal AND M8013) OR (Criticall_FaultSignal AND M8012) OR ((Normal_FaultSignal OR Criticall_FaultSignal) AND Output_NoFault);
END_PROGRAM
